// TIA Portal project "Model_Adaptive_DMC_Control" (V19)

(* hardware
DEVICE "S7-1500/ET200MP station_1"  S7-1500 station
   slot 0: "Rail_0"  Rack  6ES7 590-1***0-0AA0
   slot 1: "PLC_1"  CPU 1516-3 PN/DP  6ES7 516-3AN02-0AB0  V2.9
      slot 3: "CPU display_1"  6ES7591-1BA00-0AA0
      slot 32768: "PROFINET interface_1"  X1
         slot 32769: "Port_1"  X1 P1
         slot 32770: "Port_2"  X1 P2
      slot 33024: "PROFINET interface_2"  X2
         slot 33025: "Port_1"  X2 P1
      slot 33280: "DP interface_1"  X3
      slot 34817: "Virtual CP interface port_1"  Virtual CP interface port  Virtual CP interface port
DEVICE "Visualization"  SIMATIC PC station
   slot 0: "PC station"  Rail  SIMATIC PC-Station  V1.0
      slot 125: "Stationmanager"  Station_Manager  V6.0.4
   slot 1: "IE general_1"  IE General  IE_CP  V8.2.0
      slot 1: "PROFINET interface"  IEGeneral.Interface.8.2.0
   slot 3: "HMI_RT_1"  WinCC RT Advanced  6AV2 104-0xxxx-xxxx  17.0.0.0
      slot 33792: "Computer interface"  Host interface
*)

// ===== PLC "PLC_1"  CPU 1516-3 PN/DP =====

VAR_GLOBAL   // PLC tag table "Default tag table"
   "Tag_1" AT %M100.0 : Bool;
END_VAR

TYPE "Edge"
   STRUCT
      OneShootPositive : Bool;
      OneShootNegative : Bool;
      LastStatePositive : Bool;
      LastStateNegative : Bool;
   END_STRUCT;
END_TYPE

DATA_BLOCK "Data_DB"   // DB2
{ S7_Optimized_Access := 'FALSE' }
VERSION : 0.1
   VAR
      Manual : Int := 1;
      dOR_prev : Array[0..999] of Real;
      dOR : Real;
      dOR_max : Real := 10.0;
      "OR" : Real := 50.0;
      OR_max : Real := 100.0;
      OR_min : Real := 0.0;
      Flow : Real := 3.0;
      Flow_min : Real := 0.5;
      Flow_max : Real := 12.0;
      Power_SV_Step : Real := 10.0;
      Power_SV_Min : Real := 30.0;
      Power_SV_Max : Real := 100.0;
      Power : Real := 80.0;
      Temperature_SV_Step : Real := 10.0;
      Temperature_SV_Min : Real := 30.0;
      Temperature_SV_Max : Real := 80.0;
      Temperature_SetPoint : Real := 50.0;
      Temperature_Out : Real;
      Temperature_In : Real := 15.0;
      PWM_Period : Int := 5;
      PWM_ON : Bool;
      Heater_ON : Bool;
      Alarm_Heater : Bool;
      Alarm_Reset : Bool;
      i : Int;
      Alarm_Reset_Edge : "Edge";
      Experiment_Power : Bool;
      Experiment_Flow : Bool;
      date_time : DTL;
      start_Logging : Bool;
      Power_Nominal : Real := 12000.0;
      Density : Real := 1.0;
      Specific_Heat : Real := 4200.0;
      Volume : Real := 1.6;
      Error : Int;
   END_VAR
BEGIN
END_DATA_BLOCK

// folder: 01 Key Functions/Data_Blocks

DATA_BLOCK "Heater_PWM"   // DB3
{ S7_Optimized_Access := 'TRUE' }
VERSION : 0.1
// stored: InstanceOfName PWM
"PWM"
BEGIN
END_DATA_BLOCK

// folder: 02 Model/Data_Blocks

DATA_BLOCK "Model_Parameters_DB"   // DB7
{ S7_Optimized_Access := 'TRUE' }
VERSION : 0.1
   VAR
      x1 : Real := 15.0;
      x2 : Real;
      x3 : Real := 15.0;
      G : Real;
      tau : Real;
      delay : Int;
      k11 : Real;
      k12 : Real;
      k21 : Real;
      k22 : Real;
      k31 : Real;
      k32 : Real;
      k41 : Real;
      k42 : Real;
      y_delay : Array[0..20000] of Real;
      i : Int;
      h : Real := 0.1;
   END_VAR
BEGIN
END_DATA_BLOCK

// folder: 03 DMC Control/Data_Blocks

DATA_BLOCK "DMC_Parameters_DB"   // DB1
{ S7_Optimized_Access := 'FALSE' }
VERSION : 0.1
   VAR
      Ke : Real;
      Ku : Array[0..999] of Real;
      "max(D,N)" : Int := 347;
      D : Int := 347;
      u_subtruct : Real;
      T_before_step : Real;
   END_VAR
BEGIN
END_DATA_BLOCK

// folder: 04 Experiments/Data_Blocks

DATA_BLOCK "Experiment_Power_DB"   // DB5
{ S7_Optimized_Access := 'TRUE' }
VERSION : 0.1
// stored: InstanceOfName Experiment_Power
"Experiment_Power"
BEGIN
END_DATA_BLOCK

DATA_BLOCK "Experiment_Flow_DB"   // DB6
{ S7_Optimized_Access := 'TRUE' }
VERSION : 0.1
// stored: InstanceOfName Experiment_Flow
"Experiment_Flow"
BEGIN
END_DATA_BLOCK

// folder: (top level)

ORGANIZATION_BLOCK "Main"   // OB1, LAD, ProgramCycle
TITLE = "Main Program Sweep (Cycle)"
{ S7_Optimized_Access := 'TRUE' }
VERSION : 0.1
   VAR_INPUT
      Initial_Call : Bool;   // Initial call of this OB
      Remanence : Bool;   // =True, if remanent data are available
   END_VAR
   VAR_TEMP
      stat : Int;
   END_VAR
BEGIN

REGION Network 1: Heater control function
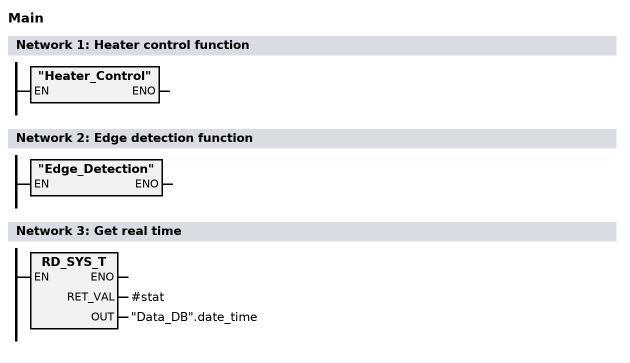
   RUNG wire#powerrail
      "Heater_Control"()
   END_RUNG
   // the same network as SCL:
   "Heater_Control"();
END_REGION

REGION Network 2: Edge detection function
   RUNG wire#powerrail
      "Edge_Detection"()
   END_RUNG
   // the same network as SCL:
   "Edge_Detection"();
END_REGION

REGION Network 3: Get real time
   #stat := RD_SYS_T(OUT => "Data_DB".date_time);
END_REGION
END_ORGANIZATION_BLOCK

ORGANIZATION_BLOCK "Startup"   // OB100, SCL, Startup
TITLE = "Complete Restart"
{ S7_Optimized_Access := 'TRUE' }
VERSION : 0.1
   VAR_INPUT
      LostRetentive : Bool;   // True if retentive data are lost
      LostRTC : Bool;   // True if date and time are lost
   END_VAR
BEGIN
   FOR "Model_Parameters_DB".i := 0 TO 19999 DO
       "Model_Parameters_DB".y_delay["Model_Parameters_DB".i] := "Data_DB".Temperature_In;
   END_FOR;

   "DMC_Parameters_DB".Ke := 0.0;
   FOR "Model_Parameters_DB".i := 0 TO 999 DO
       "DMC_Parameters_DB".Ku["Model_Parameters_DB".i] := 0.0;
   END_FOR;
END_ORGANIZATION_BLOCK

// folder: 00 Heat/Flow Control

FUNCTION "Heater_Control" : Void   // FC4, LAD
{ S7_Optimized_Access := 'TRUE' }
VERSION : 0.1
BEGIN

REGION Network 1: Request ON Heater PWM
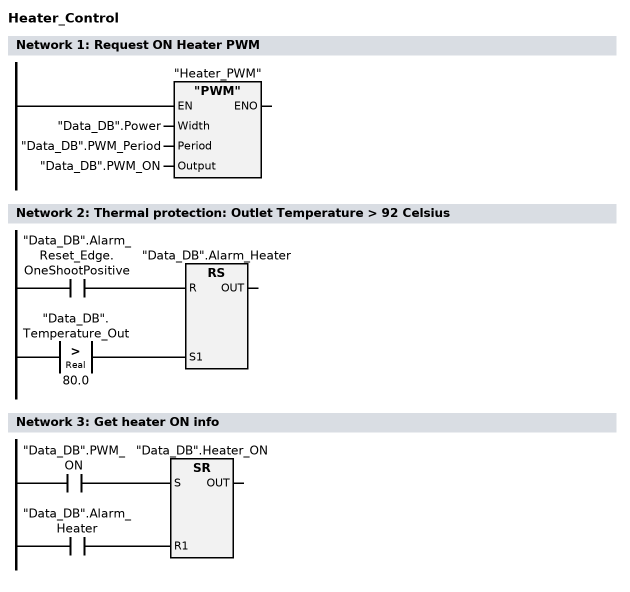
   RUNG wire#powerrail
      "Heater_PWM"(Width := "Data_DB".Power, Period := "Data_DB".PWM_Period, Output := "Data_DB".PWM_ON)
   END_RUNG
   // the same network as SCL:
   "Heater_PWM"(Width := "Data_DB".Power, Period := "Data_DB".PWM_Period, Output := "Data_DB".PWM_ON);   // "PWM"
END_REGION

REGION Network 2: Thermal protection: Outlet Temperature > 92 Celsius
   RUNG wire#powerrail
      Contact( "Data_DB".Alarm_Reset_Edge.OneShootPositive )
      S_RS(operand := "Data_DB".Alarm_Heater, s1 := wire#w1)
   END_RUNG
   RUNG wire#powerrail
      { S7_Templates := "SrcType := Real" } GT_Contact(in1 := "Data_DB".Temperature_Out, in2 := 80.0)
   END_RUNG wire#w1
   // the same network as SCL:
   IF "Data_DB".Alarm_Reset_Edge.OneShootPositive THEN
       "Data_DB".Alarm_Heater := FALSE;   // RS flip-flop
   END_IF;
   IF "Data_DB".Temperature_Out > 80.0 THEN "Data_DB".Alarm_Heater := TRUE; END_IF;
END_REGION

REGION Network 3: Get heater ON info
   RUNG wire#powerrail
      Contact( "Data_DB".PWM_ON )
      S_SR(operand := "Data_DB".Heater_ON, r1 := wire#w1)
   END_RUNG
   RUNG wire#powerrail
      Contact( "Data_DB".Alarm_Heater )
   END_RUNG wire#w1
   // the same network as SCL:
   IF "Data_DB".PWM_ON THEN
       "Data_DB".Heater_ON := TRUE;   // SR flip-flop
   END_IF;
   IF "Data_DB".Alarm_Heater THEN "Data_DB".Heater_ON := FALSE; END_IF;
END_REGION
END_FUNCTION

// folder: 01 Key Functions

FUNCTION_BLOCK "PWM"   // FB1, LAD
{ S7_Optimized_Access := 'TRUE' }
VERSION : 0.1
   VAR_INPUT
      Width : Real;
      Period : Int;   // in seconds
   END_VAR
   VAR_IN_OUT
      Output : Bool;
   END_VAR
   VAR
      Timer_PWM_ON : TON_TIME;
      Timer_PWM_OFF : TON_TIME;
   END_VAR
   VAR_TEMP
      Time_ON_Int : Int;
      Time_OFF_Int : Int;
      Time_ON : Time;
      Time_OFF : Time;
   END_VAR
BEGIN

REGION Network 1
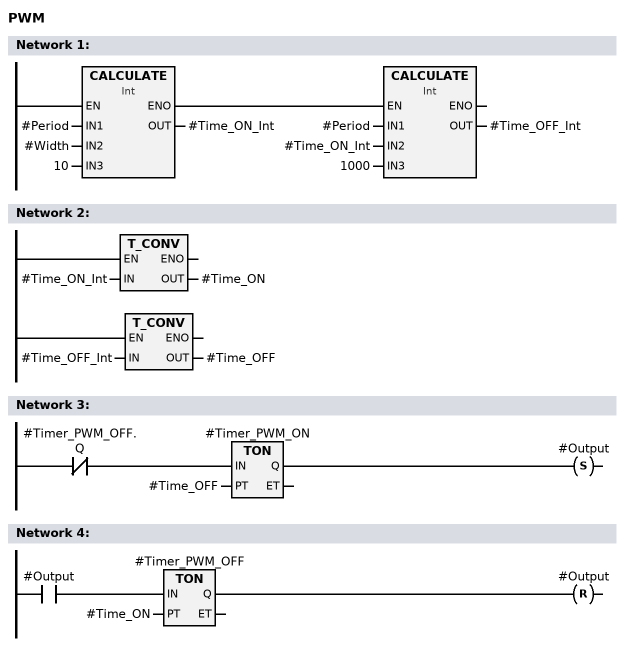
   RUNG wire#powerrail
      { S7_Templates := "SrcType := Int"; S7_Expression := "IN1*IN2*IN3" } Calculate(in1 := #Period, in2 := #Width, in3 := 10, out => #Time_ON_Int)
      { S7_Templates := "SrcType := Int"; S7_Expression := "IN1*IN3-IN2" } Calculate(in1 := #Period, in2 := #Time_ON_Int, in3 := 1000, out => #Time_OFF_Int)
   END_RUNG
   // the same network as SCL:
   #Time_ON_Int := #Period*#Width*10;
   #Time_OFF_Int := #Period*1000-#Time_ON_Int;
END_REGION

REGION Network 2
   #Time_ON := T_CONV(IN := #Time_ON_Int);
   #Time_OFF := T_CONV(IN := #Time_OFF_Int);
END_REGION

REGION Network 3
   #Timer_PWM_ON(IN := NOT #Timer_PWM_OFF.Q, PT := #Time_OFF);   // TON
   IF #Timer_PWM_ON.Q THEN #Output := TRUE; END_IF;
END_REGION

REGION Network 4
   #Timer_PWM_OFF(IN := #Output, PT := #Time_ON);   // TON
   IF #Timer_PWM_OFF.Q THEN #Output := FALSE; END_IF;
END_REGION
END_FUNCTION_BLOCK

FUNCTION "Edge_Detection" : Void   // FC2, LAD
{ S7_Optimized_Access := 'TRUE' }
VERSION : 0.1
   VAR_TEMP   // added for the SCL form of the ladder/FBD networks
      _w1 : Bool;
   END_VAR
BEGIN

REGION Network 1
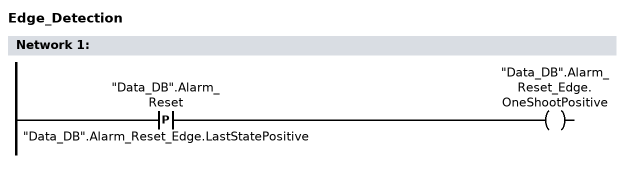
   RUNG wire#powerrail
      P_Contact(operand := "Data_DB".Alarm_Reset, bit := "Data_DB".Alarm_Reset_Edge.LastStatePositive)
      Coil( "Data_DB".Alarm_Reset_Edge.OneShootPositive )
   END_RUNG
   // the same network as SCL:
   #_w1 := "Data_DB".Alarm_Reset AND NOT "Data_DB".Alarm_Reset_Edge.LastStatePositive;   // rising edge of "Data_DB".Alarm_Reset
   "Data_DB".Alarm_Reset_Edge.LastStatePositive := "Data_DB".Alarm_Reset;
   "Data_DB".Alarm_Reset_Edge.OneShootPositive := #_w1;
END_REGION
END_FUNCTION

// folder: 02 Model

FUNCTION "StateEquationObject" : Void   // FC6, SCL
{ S7_Optimized_Access := 'TRUE' }
VERSION : 0.1
   VAR_INPUT
      x3_in : Real;
      x0 : Real;
      F : Real;
      V : Real;
      Ph : Real;
      Pnom : Real;
      cw : Real;
      ro : Real;
      h : Real;
   END_VAR
   VAR_IN_OUT
      x3_out : Real;
   END_VAR
BEGIN
   #x3_out := #h * (- #F / (60 * #V) * #x3_in + #F / (60 * #V) * #x0 + (#Ph * #Pnom) / (100 * #cw * #ro * #V));
END_FUNCTION

FUNCTION "StateEquationSensor" : Void   // FC7, SCL
{ S7_Optimized_Access := 'TRUE' }
VERSION : 0.1
   VAR_INPUT
      x1_in : Real;
      x2_in : Real;
      P : Real;
      G : Real;
      tau : Real;
      h : Real;
   END_VAR
   VAR_IN_OUT
      x1_out : Real;
      x2_out : Real;
   END_VAR
BEGIN

   #x1_out := #h * #x2_in;
   #x2_out := #h * (-2 / #tau * #x2_in - 1 / (#tau ** 2) * #x1_in + #G * #P / (#tau ** 2));
END_FUNCTION

ORGANIZATION_BLOCK "Model"   // OB30, SCL, CyclicInterrupt
{ S7_Optimized_Access := 'TRUE' }
VERSION : 0.1
   VAR_INPUT
      Initial_Call : Bool;   // Initial call of this OB
      Event_Count : Int;   // Events discarded
   END_VAR
   VAR_TEMP
      temp_PWM_ON : Real;
   END_VAR
BEGIN
   "Data_DB".Flow := "Data_DB"."OR" * "Data_DB".Flow_max / 100;

   IF "Data_DB".Flow < "Data_DB".Flow_min THEN
       "Data_DB".Flow := "Data_DB".Flow_min;
   END_IF;

   "Model_Parameters_DB".G := -0.0002347 * "Data_DB".Power + 1.012;
   "Model_Parameters_DB".tau := 19.08 * "Data_DB".Flow ** (-0.4293) - 4.042;
   "Model_Parameters_DB".delay := CEIL((11.93 * "Data_DB".Flow ** (-0.78) + 2.73)/"Model_Parameters_DB".h);

   //IF "Data_DB".PWM_ON THEN
   //    #temp_PWM_ON := 100;
   //END_IF;

   "StateEquationObject"(x3_in:="Model_Parameters_DB".x3,
                         x0:="Data_DB".Temperature_In,
                         F:="Data_DB".Flow,
                         V:="Data_DB".Volume,
                         Ph:="Data_DB".Power,
                         Pnom:="Data_DB".Power_Nominal,
                         cw:="Data_DB".Specific_Heat,
                         ro:="Data_DB".Density,
                         h:="Model_Parameters_DB".h,
                         x3_out:="Model_Parameters_DB".k11);
   "StateEquationObject"(x3_in:="Model_Parameters_DB".x3 + 0.5*"Model_Parameters_DB".k11,
                         x0:="Data_DB".Temperature_In,
                         F:="Data_DB".Flow,
                         V:="Data_DB".Volume,
                         Ph:="Data_DB".Power,
                         Pnom:="Data_DB".Power_Nominal,
                         cw:="Data_DB".Specific_Heat,
                         ro:="Data_DB".Density,
                         h:="Model_Parameters_DB".h,
                         x3_out:="Model_Parameters_DB".k21);
   "StateEquationObject"(x3_in:="Model_Parameters_DB".x3 + 0.5*"Model_Parameters_DB".k21,
                         x0:="Data_DB".Temperature_In,
                         F:="Data_DB".Flow,
                         V:="Data_DB".Volume,
                         Ph:="Data_DB".Power,
                         Pnom:="Data_DB".Power_Nominal,
                         cw:="Data_DB".Specific_Heat,
                         ro:="Data_DB".Density,
                         h:="Model_Parameters_DB".h,
                         x3_out:="Model_Parameters_DB".k31);
   "StateEquationObject"(x3_in:="Model_Parameters_DB".x3 + "Model_Parameters_DB".k31,
                         x0:="Data_DB".Temperature_In,
                         F:="Data_DB".Flow,
                         V:="Data_DB".Volume,
                         Ph:="Data_DB".Power,
                         Pnom:="Data_DB".Power_Nominal,
                         cw:="Data_DB".Specific_Heat,
                         ro:="Data_DB".Density,
                         h:="Model_Parameters_DB".h,
                         x3_out:="Model_Parameters_DB".k41);

   "Model_Parameters_DB".x3 := "Model_Parameters_DB".x3 + ("Model_Parameters_DB".k11 + 2.0 * "Model_Parameters_DB".k21 + 2.0 * "Model_Parameters_DB".k31 + "Model_Parameters_DB".k41) / 6.0;

   "StateEquationSensor"(x1_in:="Model_Parameters_DB".x1,
                         x2_in:="Model_Parameters_DB".x2,
                         P:="Model_Parameters_DB".x3,
                         G:="Model_Parameters_DB".G,
                         tau:="Model_Parameters_DB".tau,
                         h:="Model_Parameters_DB".h,
                         x1_out:="Model_Parameters_DB".k11,
                         x2_out:="Model_Parameters_DB".k12);
   "StateEquationSensor"(x1_in:="Model_Parameters_DB".x1 + 0.5*"Model_Parameters_DB".k11,
                         x2_in:="Model_Parameters_DB".x2 + 0.5*"Model_Parameters_DB".k12,
                         P:="Model_Parameters_DB".x3,
                         G:="Model_Parameters_DB".G,
                         tau:="Model_Parameters_DB".tau,
                         h:="Model_Parameters_DB".h,
                         x1_out:="Model_Parameters_DB".k21,
                         x2_out:="Model_Parameters_DB".k22);
   "StateEquationSensor"(x1_in:="Model_Parameters_DB".x1 + 0.5*"Model_Parameters_DB".k21,
                         x2_in:="Model_Parameters_DB".x2 + 0.5*"Model_Parameters_DB".k22,
                         P:="Model_Parameters_DB".x3,
                         G:="Model_Parameters_DB".G,
                         tau:="Model_Parameters_DB".tau,
                         h:="Model_Parameters_DB".h,
                         x1_out:="Model_Parameters_DB".k31,
                         x2_out:="Model_Parameters_DB".k32);
   "StateEquationSensor"(x1_in:="Model_Parameters_DB".x1 + "Model_Parameters_DB".k31,
                         x2_in:="Model_Parameters_DB".x2 + "Model_Parameters_DB".k32,
                         P:="Model_Parameters_DB".x3,
                         G:="Model_Parameters_DB".G,
                         tau:="Model_Parameters_DB".tau,
                         h:="Model_Parameters_DB".h,
                         x1_out:="Model_Parameters_DB".k41,
                         x2_out:="Model_Parameters_DB".k42);

   "Model_Parameters_DB".x1 := "Model_Parameters_DB".x1 + ("Model_Parameters_DB".k11 + 2.0 * "Model_Parameters_DB".k21 + 2.0 * "Model_Parameters_DB".k31 + "Model_Parameters_DB".k41) / 6.0;
   "Model_Parameters_DB".x2 := "Model_Parameters_DB".x2 + ("Model_Parameters_DB".k12 + 2.0 * "Model_Parameters_DB".k22 + 2.0 * "Model_Parameters_DB".k32 + "Model_Parameters_DB".k42) / 6.0;

   FOR "Model_Parameters_DB".i := 0 TO 200 DO
       "Model_Parameters_DB".y_delay["Model_Parameters_DB".delay + "Model_Parameters_DB".i] := "Model_Parameters_DB".x1;
   END_FOR;
   "Data_DB".Temperature_Out := "Model_Parameters_DB".y_delay[0];

   FOR "Model_Parameters_DB".i := 0 TO "Model_Parameters_DB".delay - 1 DO
       "Model_Parameters_DB".y_delay["Model_Parameters_DB".i] := "Model_Parameters_DB".y_delay["Model_Parameters_DB".i + 1];
   END_FOR;
END_ORGANIZATION_BLOCK

// folder: 03 DMC Control

ORGANIZATION_BLOCK "DMC_Control"   // OB31, SCL, CyclicInterrupt
{ S7_Optimized_Access := 'TRUE' }
VERSION : 0.1
   VAR_INPUT
      Initial_Call : Bool;   // Initial call of this OB
      Event_Count : Int;   // Events discarded
   END_VAR
   VAR_TEMP
      temp_Temperature_Setpoint : Real;
      temp_u_subtruct : Real;
      temp_Power_Normalization : Real;
   END_VAR
BEGIN
   IF "Data_DB".Manual = 0 THEN
       // Calculate needed power change
       "DMC_Parameters_DB".u_subtruct := 0.0;
       FOR "Data_DB".i := 0 TO "DMC_Parameters_DB".D - 1 DO
           "DMC_Parameters_DB".u_subtruct := "DMC_Parameters_DB".u_subtruct + "DMC_Parameters_DB".Ku["Data_DB".i] * "Data_DB".dOR_prev["Data_DB".i];
       END_FOR;

       "Data_DB".dOR := "DMC_Parameters_DB".Ke * ("Data_DB".Temperature_SetPoint - "Data_DB".Temperature_Out) - "DMC_Parameters_DB".u_subtruct;

       IF "Data_DB".dOR > "Data_DB".dOR_max THEN
           "Data_DB".dOR := "Data_DB".dOR_max;
       ELSIF "Data_DB".dOR < - "Data_DB".dOR_max THEN
           "Data_DB".dOR := - "Data_DB".dOR_max;
       END_IF;

       // Put current power change to the vector of previous power changes
       FOR "Data_DB".i := "DMC_Parameters_DB".D - 1 TO 1 BY -1 DO
           "Data_DB".dOR_prev["Data_DB".i] := "Data_DB".dOR_prev["Data_DB".i - 1];
       END_FOR;
       "Data_DB".dOR_prev[0] := "Data_DB".dOR;

       // Calculate current power
       "Data_DB"."OR" := "Data_DB"."OR" + "Data_DB".dOR;

       IF "Data_DB"."OR" > "Data_DB".OR_max THEN
           "Data_DB"."OR" := "Data_DB".OR_max;
       ELSIF "Data_DB"."OR" < "Data_DB".OR_min THEN
           "Data_DB"."OR" := "Data_DB".OR_min;
       END_IF;
   END_IF;
END_ORGANIZATION_BLOCK

// folder: 04 Experiments

FUNCTION_BLOCK "Experiment_Power"   // FB2, LAD
{ S7_Optimized_Access := 'TRUE' }
VERSION : 0.1
   VAR_IN_OUT
      Experiment_Permission : Bool;
      Power : Real;
      Flow : Real;
   END_VAR
   VAR
      State : Int;
      IEC_Timer_0_Instance : TON_TIME;
      IEC_Timer_0_Instance_1 : TON_TIME;
      IEC_Timer_0_Instance_2 : TON_TIME;
      IEC_Timer_0_Instance_3 : TON_TIME;
      IEC_Timer_0_Instance_4 : TON_TIME;
      IEC_Timer_0_Instance_5 : TON_TIME;
      IEC_Timer_0_Instance_6 : TON_TIME;
      IEC_Timer_0_Instance_7 : TON_TIME;
      IEC_Timer_0_Instance_8 : TON_TIME;
      IEC_Timer_0_Instance_9 : TON_TIME;
      IEC_Timer_0_Instance_10 : TON_TIME;
      IEC_Timer_0_Instance_11 : TON_TIME;
      IEC_Timer_0_Instance_12 : TON_TIME;
      IEC_Timer_0_Instance_13 : TON_TIME;
      IEC_Timer_0_Instance_14 : TON_TIME;
   END_VAR
   VAR_TEMP   // added for the SCL form of the ladder/FBD networks
      _w1 : Bool;
   END_VAR
BEGIN

REGION Network 1
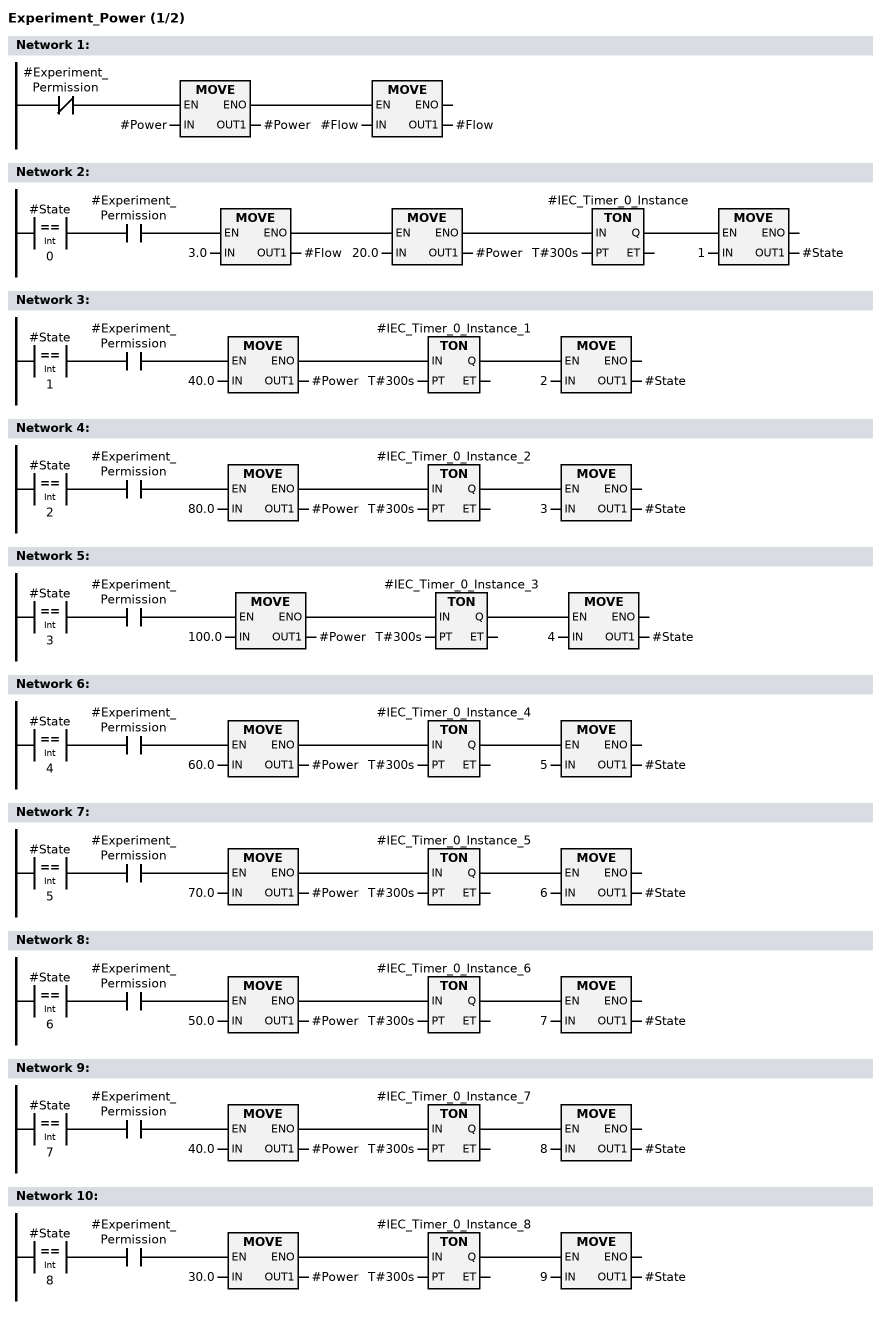
   RUNG wire#powerrail
      I_Contact( #Experiment_Permission )
      Move(in := #Power, out1 => #Power)
      Move(in := #Flow, out1 => #Flow)
   END_RUNG
   // the same network as SCL:
   IF NOT #Experiment_Permission THEN
       #Power := #Power;
       #Flow := #Flow;
   END_IF;
END_REGION

REGION Network 2
   #_w1 := (#State = 0) AND #Experiment_Permission;
   IF #_w1 THEN
       #Flow := 3.0;
       #Power := 20.0;
   END_IF;
   #IEC_Timer_0_Instance(IN := #_w1, PT := T#300s);   // TON
   IF #IEC_Timer_0_Instance.Q THEN #State := 1; END_IF;
END_REGION

REGION Network 3
   #_w1 := (#State = 1) AND #Experiment_Permission;
   IF #_w1 THEN #Power := 40.0; END_IF;
   #IEC_Timer_0_Instance_1(IN := #_w1, PT := T#300s);   // TON
   IF #IEC_Timer_0_Instance_1.Q THEN #State := 2; END_IF;
END_REGION

REGION Network 4
   #_w1 := (#State = 2) AND #Experiment_Permission;
   IF #_w1 THEN #Power := 80.0; END_IF;
   #IEC_Timer_0_Instance_2(IN := #_w1, PT := T#300s);   // TON
   IF #IEC_Timer_0_Instance_2.Q THEN #State := 3; END_IF;
END_REGION

REGION Network 5
   #_w1 := (#State = 3) AND #Experiment_Permission;
   IF #_w1 THEN #Power := 100.0; END_IF;
   #IEC_Timer_0_Instance_3(IN := #_w1, PT := T#300s);   // TON
   IF #IEC_Timer_0_Instance_3.Q THEN #State := 4; END_IF;
END_REGION

REGION Network 6
   #_w1 := (#State = 4) AND #Experiment_Permission;
   IF #_w1 THEN #Power := 60.0; END_IF;
   #IEC_Timer_0_Instance_4(IN := #_w1, PT := T#300s);   // TON
   IF #IEC_Timer_0_Instance_4.Q THEN #State := 5; END_IF;
END_REGION

REGION Network 7
   #_w1 := (#State = 5) AND #Experiment_Permission;
   IF #_w1 THEN #Power := 70.0; END_IF;
   #IEC_Timer_0_Instance_5(IN := #_w1, PT := T#300s);   // TON
   IF #IEC_Timer_0_Instance_5.Q THEN #State := 6; END_IF;
END_REGION

REGION Network 8
   #_w1 := (#State = 6) AND #Experiment_Permission;
   IF #_w1 THEN #Power := 50.0; END_IF;
   #IEC_Timer_0_Instance_6(IN := #_w1, PT := T#300s);   // TON
   IF #IEC_Timer_0_Instance_6.Q THEN #State := 7; END_IF;
END_REGION

REGION Network 9
   #_w1 := (#State = 7) AND #Experiment_Permission;
   IF #_w1 THEN #Power := 40.0; END_IF;
   #IEC_Timer_0_Instance_7(IN := #_w1, PT := T#300s);   // TON
   IF #IEC_Timer_0_Instance_7.Q THEN #State := 8; END_IF;
END_REGION

REGION Network 10
   #_w1 := (#State = 8) AND #Experiment_Permission;
   IF #_w1 THEN #Power := 30.0; END_IF;
   #IEC_Timer_0_Instance_8(IN := #_w1, PT := T#300s);   // TON
   IF #IEC_Timer_0_Instance_8.Q THEN #State := 9; END_IF;
END_REGION

REGION Network 11
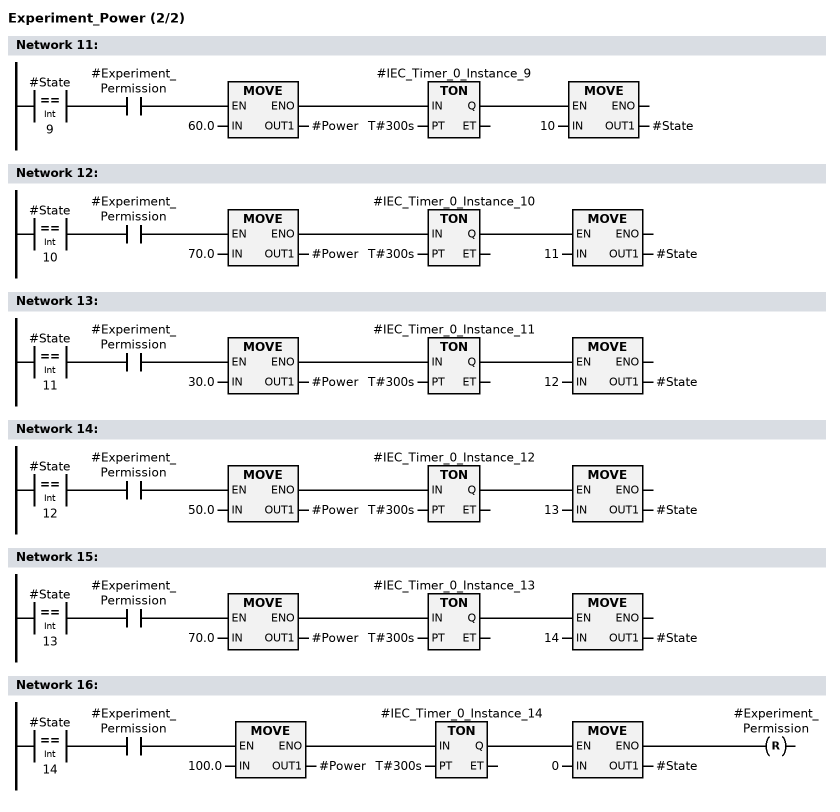
   #_w1 := (#State = 9) AND #Experiment_Permission;
   IF #_w1 THEN #Power := 60.0; END_IF;
   #IEC_Timer_0_Instance_9(IN := #_w1, PT := T#300s);   // TON
   IF #IEC_Timer_0_Instance_9.Q THEN #State := 10; END_IF;
END_REGION

REGION Network 12
   #_w1 := (#State = 10) AND #Experiment_Permission;
   IF #_w1 THEN #Power := 70.0; END_IF;
   #IEC_Timer_0_Instance_10(IN := #_w1, PT := T#300s);   // TON
   IF #IEC_Timer_0_Instance_10.Q THEN #State := 11; END_IF;
END_REGION

REGION Network 13
   #_w1 := (#State = 11) AND #Experiment_Permission;
   IF #_w1 THEN #Power := 30.0; END_IF;
   #IEC_Timer_0_Instance_11(IN := #_w1, PT := T#300s);   // TON
   IF #IEC_Timer_0_Instance_11.Q THEN #State := 12; END_IF;
END_REGION

REGION Network 14
   #_w1 := (#State = 12) AND #Experiment_Permission;
   IF #_w1 THEN #Power := 50.0; END_IF;
   #IEC_Timer_0_Instance_12(IN := #_w1, PT := T#300s);   // TON
   IF #IEC_Timer_0_Instance_12.Q THEN #State := 13; END_IF;
END_REGION

REGION Network 15
   #_w1 := (#State = 13) AND #Experiment_Permission;
   IF #_w1 THEN #Power := 70.0; END_IF;
   #IEC_Timer_0_Instance_13(IN := #_w1, PT := T#300s);   // TON
   IF #IEC_Timer_0_Instance_13.Q THEN #State := 14; END_IF;
END_REGION

REGION Network 16
   #_w1 := (#State = 14) AND #Experiment_Permission;
   IF #_w1 THEN #Power := 100.0; END_IF;
   #IEC_Timer_0_Instance_14(IN := #_w1, PT := T#300s);   // TON
   IF #IEC_Timer_0_Instance_14.Q THEN
       #State := 0;
       #Experiment_Permission := FALSE;
   END_IF;
END_REGION
END_FUNCTION_BLOCK

FUNCTION_BLOCK "Experiment_Flow"   // FB3, LAD
{ S7_Optimized_Access := 'TRUE' }
VERSION : 0.1
   VAR_IN_OUT
      Experiment_Permission : Bool;
      Power : Real;
      Flow : Real;
   END_VAR
   VAR
      State : Int;
      IEC_Timer_0_Instance : TON_TIME;
      IEC_Timer_0_Instance_1 : TON_TIME;
      IEC_Timer_0_Instance_2 : TON_TIME;
      IEC_Timer_0_Instance_3 : TON_TIME;
      IEC_Timer_0_Instance_4 : TON_TIME;
      IEC_Timer_0_Instance_5 : TON_TIME;
      IEC_Timer_0_Instance_6 : TON_TIME;
      IEC_Timer_0_Instance_7 : TON_TIME;
      IEC_Timer_0_Instance_8 : TON_TIME;
      IEC_Timer_0_Instance_9 : TON_TIME;
      IEC_Timer_0_Instance_10 : TON_TIME;
      IEC_Timer_0_Instance_11 : TON_TIME;
      IEC_Timer_0_Instance_12 : TON_TIME;
      IEC_Timer_0_Instance_13 : TON_TIME;
      IEC_Timer_0_Instance_14 : TON_TIME;
   END_VAR
   VAR_TEMP   // added for the SCL form of the ladder/FBD networks
      _w1 : Bool;
   END_VAR
BEGIN

REGION Network 1
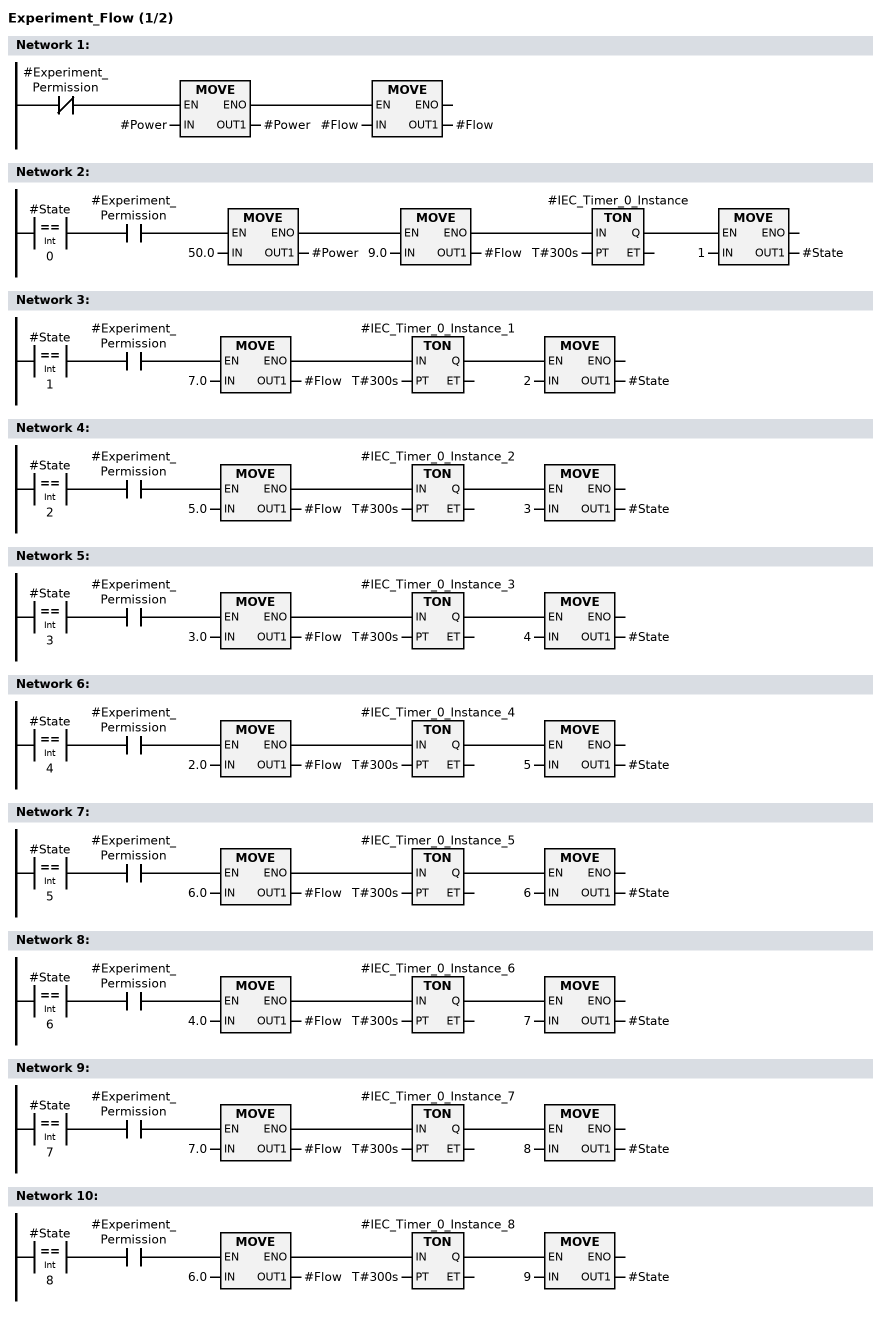
   RUNG wire#powerrail
      I_Contact( #Experiment_Permission )
      Move(in := #Power, out1 => #Power)
      Move(in := #Flow, out1 => #Flow)
   END_RUNG
   // the same network as SCL:
   IF NOT #Experiment_Permission THEN
       #Power := #Power;
       #Flow := #Flow;
   END_IF;
END_REGION

REGION Network 2
   #_w1 := (#State = 0) AND #Experiment_Permission;
   IF #_w1 THEN
       #Power := 50.0;
       #Flow := 9.0;
   END_IF;
   #IEC_Timer_0_Instance(IN := #_w1, PT := T#300s);   // TON
   IF #IEC_Timer_0_Instance.Q THEN #State := 1; END_IF;
END_REGION

REGION Network 3
   #_w1 := (#State = 1) AND #Experiment_Permission;
   IF #_w1 THEN #Flow := 7.0; END_IF;
   #IEC_Timer_0_Instance_1(IN := #_w1, PT := T#300s);   // TON
   IF #IEC_Timer_0_Instance_1.Q THEN #State := 2; END_IF;
END_REGION

REGION Network 4
   #_w1 := (#State = 2) AND #Experiment_Permission;
   IF #_w1 THEN #Flow := 5.0; END_IF;
   #IEC_Timer_0_Instance_2(IN := #_w1, PT := T#300s);   // TON
   IF #IEC_Timer_0_Instance_2.Q THEN #State := 3; END_IF;
END_REGION

REGION Network 5
   #_w1 := (#State = 3) AND #Experiment_Permission;
   IF #_w1 THEN #Flow := 3.0; END_IF;
   #IEC_Timer_0_Instance_3(IN := #_w1, PT := T#300s);   // TON
   IF #IEC_Timer_0_Instance_3.Q THEN #State := 4; END_IF;
END_REGION

REGION Network 6
   #_w1 := (#State = 4) AND #Experiment_Permission;
   IF #_w1 THEN #Flow := 2.0; END_IF;
   #IEC_Timer_0_Instance_4(IN := #_w1, PT := T#300s);   // TON
   IF #IEC_Timer_0_Instance_4.Q THEN #State := 5; END_IF;
END_REGION

REGION Network 7
   #_w1 := (#State = 5) AND #Experiment_Permission;
   IF #_w1 THEN #Flow := 6.0; END_IF;
   #IEC_Timer_0_Instance_5(IN := #_w1, PT := T#300s);   // TON
   IF #IEC_Timer_0_Instance_5.Q THEN #State := 6; END_IF;
END_REGION

REGION Network 8
   #_w1 := (#State = 6) AND #Experiment_Permission;
   IF #_w1 THEN #Flow := 4.0; END_IF;
   #IEC_Timer_0_Instance_6(IN := #_w1, PT := T#300s);   // TON
   IF #IEC_Timer_0_Instance_6.Q THEN #State := 7; END_IF;
END_REGION

REGION Network 9
   #_w1 := (#State = 7) AND #Experiment_Permission;
   IF #_w1 THEN #Flow := 7.0; END_IF;
   #IEC_Timer_0_Instance_7(IN := #_w1, PT := T#300s);   // TON
   IF #IEC_Timer_0_Instance_7.Q THEN #State := 8; END_IF;
END_REGION

REGION Network 10
   #_w1 := (#State = 8) AND #Experiment_Permission;
   IF #_w1 THEN #Flow := 6.0; END_IF;
   #IEC_Timer_0_Instance_8(IN := #_w1, PT := T#300s);   // TON
   IF #IEC_Timer_0_Instance_8.Q THEN #State := 9; END_IF;
END_REGION

REGION Network 11
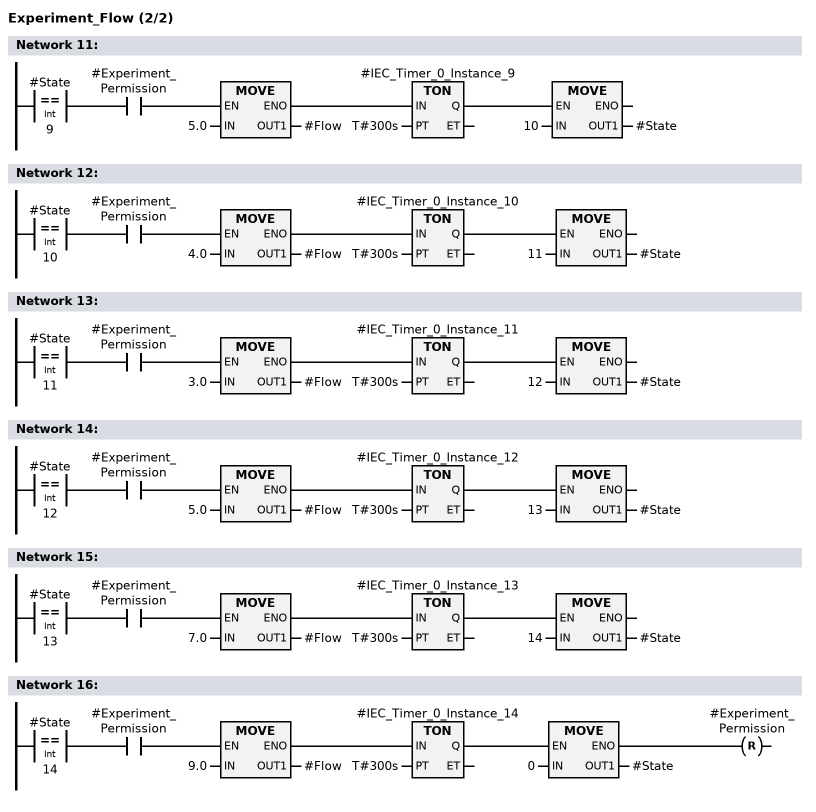
   #_w1 := (#State = 9) AND #Experiment_Permission;
   IF #_w1 THEN #Flow := 5.0; END_IF;
   #IEC_Timer_0_Instance_9(IN := #_w1, PT := T#300s);   // TON
   IF #IEC_Timer_0_Instance_9.Q THEN #State := 10; END_IF;
END_REGION

REGION Network 12
   #_w1 := (#State = 10) AND #Experiment_Permission;
   IF #_w1 THEN #Flow := 4.0; END_IF;
   #IEC_Timer_0_Instance_10(IN := #_w1, PT := T#300s);   // TON
   IF #IEC_Timer_0_Instance_10.Q THEN #State := 11; END_IF;
END_REGION

REGION Network 13
   #_w1 := (#State = 11) AND #Experiment_Permission;
   IF #_w1 THEN #Flow := 3.0; END_IF;
   #IEC_Timer_0_Instance_11(IN := #_w1, PT := T#300s);   // TON
   IF #IEC_Timer_0_Instance_11.Q THEN #State := 12; END_IF;
END_REGION

REGION Network 14
   #_w1 := (#State = 12) AND #Experiment_Permission;
   IF #_w1 THEN #Flow := 5.0; END_IF;
   #IEC_Timer_0_Instance_12(IN := #_w1, PT := T#300s);   // TON
   IF #IEC_Timer_0_Instance_12.Q THEN #State := 13; END_IF;
END_REGION

REGION Network 15
   #_w1 := (#State = 13) AND #Experiment_Permission;
   IF #_w1 THEN #Flow := 7.0; END_IF;
   #IEC_Timer_0_Instance_13(IN := #_w1, PT := T#300s);   // TON
   IF #IEC_Timer_0_Instance_13.Q THEN #State := 14; END_IF;
END_REGION

REGION Network 16
   #_w1 := (#State = 14) AND #Experiment_Permission;
   IF #_w1 THEN #Flow := 9.0; END_IF;
   #IEC_Timer_0_Instance_14(IN := #_w1, PT := T#300s);   // TON
   IF #IEC_Timer_0_Instance_14.Q THEN
       #State := 0;
       #Experiment_Permission := FALSE;
   END_IF;
END_REGION
END_FUNCTION_BLOCK

(* ===== HMI "HMI_RT_1" =====
connection "HMI_Connection_1": ETHERNET, S7_1500_OMS

HMI tags "Default tag table"
   "count_Logs" : DInt, internal
   "start_Logging" : Bool = PLC Data_DB.start_Logging AT %DB2.DBX4096.0, 100 ms
   "Alarm_Heater" : Bool = PLC Data_DB.Alarm_Heater AT %DB2.DBX4076.2, 100 ms
   "Alarm_Reset" : Bool = PLC Data_DB.Alarm_Reset AT %DB2.DBX4076.3, 100 ms
   "Temperature_Setpoint" : Real = PLC Data_DB.Temperature_SetPoint AT %DB2.DBD4062, 100 ms
   "OR" : Real = PLC Data_DB.OR AT %DB2.DBD4010, 100 ms
   "Power" : Real = PLC Data_DB.Power AT %DB2.DBD4046, 100 ms
   "Temperature_In" : Real = PLC Data_DB.Temperature_In AT %DB2.DBD4070, 100 ms
   "Temperature_Out" : Real = PLC Data_DB.Temperature_Out AT %DB2.DBD4066, 100 ms
   "Heater_ON" : Bool = PLC Data_DB.Heater_ON AT %DB2.DBX4076.1, 100 ms
   "PWM_Period" : Int = PLC Data_DB.PWM_Period AT %DB2.DBW4074, 100 ms
   "Time" : DTL = PLC Data_DB.date_time AT %DB2.DBX4084.0, 100 ms
   "Flow" : Real = PLC Data_DB.Flow AT %DB2.DBD4022, 100 ms
   "Temperature_SV_Step" : Real = PLC Data_DB.Temperature_SV_Step AT %DB2.DBD4050, 1 s
   "Temperature_SV_Min" : Real = PLC Data_DB.Temperature_SV_Min AT %DB2.DBD4054, 1 s
   "Temperature_SV_Max" : Real = PLC Data_DB.Temperature_SV_Max AT %DB2.DBD4058, 1 s
   "Power_SV_Step" : Real = PLC Data_DB.Power_SV_Step AT %DB2.DBD4034, 1 s
   "Power_SV_Min" : Real = PLC Data_DB.Power_SV_Min AT %DB2.DBD4038, 1 s
   "Power_SV_Max" : Real = PLC Data_DB.Power_SV_Max AT %DB2.DBD4042, 1 s
   "Manual" : Int = PLC Data_DB.Manual AT %DB2.DBW0, 1 s

VB script "csv_export"
   Dim FolderPath, ObjectPath, Filename, File, FileExist, Columns, Row, toogle
   
   
   toogle=SmartTags("start_Logging")
   'SmartTags("test")=toogle
   
   If  toogle <> 0 Then
   	
   	count_Logs = count_Logs+1
   	
   
   	'FolderPath = "C:\_DOC\"
   	FolderPath = "C:\Users\Gabriel\OneDrive\Desktop\Model-Predictive-Control\Data\"
   
   	Filename = "Model_Verification.csv"
   
   	Set ObjectPath = CreateObject("Scripting.FilesystemObject")
   
   	'Check if folder exists
   
   	If Not ObjectPath.FolderExists(FolderPath) Then              
   
   		ObjectPath.CreateFolder FolderPath     
   
   	End If
   
   	' Check if file exists
   
   	Set File = CreateObject("Scripting.FilesystemObject")
   
   	FileExist = File.FileExists(FolderPath & "\" & Filename)
   
   	If FileExist = False Then
   
   		File.CreateTextFile(FolderPath & "\" & Filename)
   
   		Set Columns = File.OpenTextFile(FolderPath & "\" & Filename, 8)
   
                 	'Columns.WriteLine("Data1 ; Data2 ; Data3")
   				'Columns.WriteLine("time; F1; F2; F3; power_duzy_piec; PWM_duzy_piec; power_maly_piec; PWM_maly_piec; Tin_piec;Tour_piec; Tin_maly_piec; Tout_maly_piec; Tin_wym_dol_ciepla; Tin_wym_dol_zimna; Tout_wym_dol_ciepla; Tout_wym_dol_zimna; Tin_wym_gora_ciepla; Tin_wym_gora_zimna; Tout_wym_gora_ciepla; Tout_wym_gora_zimna; Pin_instalacja; Pin_wym_gora_ciepla; Pin_wym_gora_zmina; Pout_wym_gora_ciepla; Pout_wym_gora_zimna; P_PZ2; P_PZ3; T_otoczenia; Zmienne_PID_F1_SP; F1_SP; F2_SP; F3_SP")
                   Columns.WriteLine("Time; Flow; Power; Temperature_Setpoint; Temperature_In; Temperature_Out; Pressure_In; Flow_Setpoint")
                   Columns.Close                 
   
                   Set File = Nothing           
   
   	End If
   
   
   
   	'Write data to file
   
   	Set File = CreateObject("Scripting.FilesystemObject")
   
   	Set Row = File.OpenTextFile(FolderPath & "\" & Filename, 8)
   
   
   	'Row.WriteLine(SmartTags("F1_SP") & ";" & SmartTags("F2_SP") & ";" & SmartTags("F3_SP") & ";")
   	Row.WriteLine(SmartTags("Time")& ";" &SmartTags("OR")& ";" &SmartTags("Power")& ";" &SmartTags("Temperature_Setpoint")& ";" &SmartTags("Temperature_In")& ";" &SmartTags("Temperature_Out")& ";" &SmartTags("Pressure_In")& ";" &SmartTags("Flow_Setpoint"))
   	
   	Row.Close
   
   	Set File = Nothing  'Here we are releasing the File.
   End If
*)